TYPE ST_InfoDataConnection :
STRUCT
	usiMapState:USINT;
	usiMapDiag:USINT;
	bySignals:BYTE;
END_STRUCT
END_TYPE

(* stored: Version 1.1.0.1, ProductVersion 3.1.0.20
   DUT ST_InfoDataConnection: Id {bf62ba12-1126-4e78-a43d-9d3456d178c3} *)
